FUNCTION_BLOCK SmallSortingConveyor EXTENDS Conveyor
VAR_INPUT
END_VAR
VAR_OUTPUT
END_VAR
VAR
	//Sensors
	m_PresencesensorStart : PresenceSensor;
	m_PresencesensorEnd : PresenceSensor;
	m_Opticalsensor : OpticalSensor;
	m_Inductivesensor : InductiveSensor;
	
	//Ramps
	m_Ramp : Ramp;
	
	//Pusher
	m_Switch : Switch;
END_VAR

PROPERTY LightWPAtMid : BOOL
GET
LightWPAtMid := m_Opticalsensor.Value;
END_GET
END_PROPERTY

PROPERTY MetalWPAtMid : BOOL
GET
MetalWPAtMid := m_Inductivesensor.Value;
END_GET
END_PROPERTY

METHOD METH_Switch_Extend : BOOL
VAR_INPUT
END_VAR
m_Switch.METH_Extend();
END_METHOD

METHOD METH_Switch_Retract : BOOL
VAR_INPUT
END_VAR
m_Switch.METH_Retract();
END_METHOD

PROPERTY WPAtEnd : BOOL
GET
WPAtEnd := m_PresencesensorEnd.Value;
END_GET
END_PROPERTY

PROPERTY WPAtRampEnd : BOOL
GET
WPAtRampEnd := m_Ramp.m_presenceSensorRampFull.Value;
END_GET
END_PROPERTY

PROPERTY WPAtStart : BOOL
GET
WPAtStart := m_PresencesensorStart.Value;
END_GET
END_PROPERTY

END_FUNCTION_BLOCK

(* stored: Version 1.1.0.1, ProductVersion 3.1.4024.4
   POU SmallSortingConveyor: Id {3714cf9c-d595-4df3-b202-737827676521}, SpecialFunc None
   Folder Methods: Id {f24fd5c1-477f-40e5-b1d2-5905ffa33485}
   Folder Properties: Id {8679b29f-ab4d-421f-96ec-3eaabb4bb3fe}
   Property LightWPAtMid: Id {2237b367-9b7e-431e-834e-93e0d5ba7ecb}
   Get Get: Id {1767380a-69e5-41cf-aa15-8e7ff8460a60}
   Property MetalWPAtMid: Id {5e56331b-00dd-4845-8d03-e2e236ba54f6}
   Get Get: Id {75551164-3756-46ad-b077-08017d91948f}
   Method METH_Switch_Extend: Id {9b7390ad-8e73-4fa1-99f2-ba73faca2a81}
   Method METH_Switch_Retract: Id {bbd0f736-fce1-418f-9af3-4a30e5e1b131}
   Property WPAtEnd: Id {1f6208e9-1151-414e-b259-e1b5ebcb9d58}
   Get Get: Id {c922685e-6228-46ff-8499-ecc54fe65e99}
   Property WPAtRampEnd: Id {8d168ced-2bc9-4b6c-97b5-6c52d31b49f2}
   Get Get: Id {7ccb546a-5e86-4bca-8d46-ab3fe066bc38}
   Property WPAtStart: Id {75340cc2-2a98-4d7a-a7ed-611102ffbd2c}
   Get Get: Id {4d6ab26d-9774-4d9d-9a5c-75ea669f7a89} *)
